FUNCTION F_TMO_RoughVRC : BOOL
VAR_INPUT
END_VAR
VAR
END_VAR

END_FUNCTION

(* stored: Version 1.1.0.1, ProductVersion 3.1.4022.18
   POU F_TMO_RoughVRC: Id {923fd527-01a5-4fc8-9fca-a16621757af1}, SpecialFunc None *)
